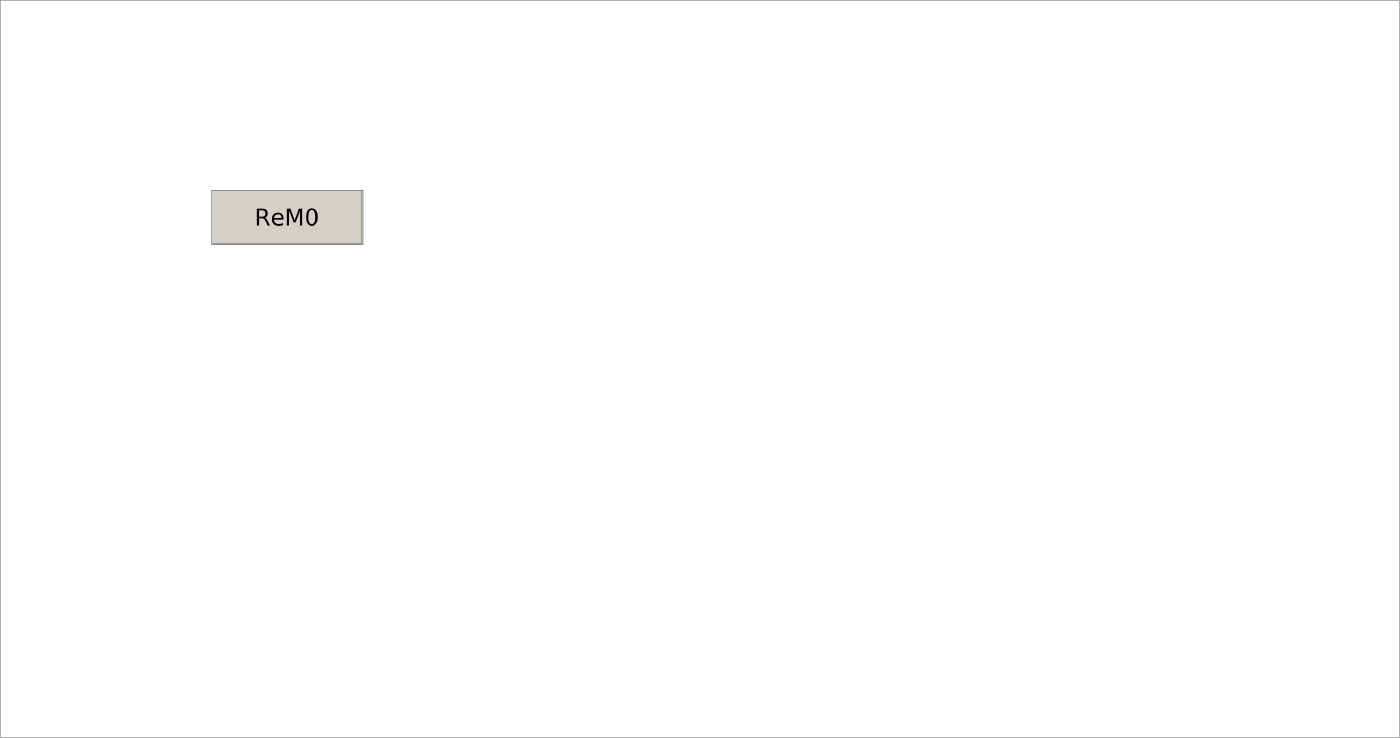
VISUALIZATION visu_Others  // 2048x1080
    Button (309,278 222x80), "ReM0", colour toggle: G_HMI.iReM =0
        p573394764: 16#FF00FF00
        OnMouseDown: execute { G_HMI.iReM  := 0; G_HMI.iMainFrame	:= 0; }
END_VISUALIZATION

(* stored: Version 1.1.0.1, ProductVersion 3.1.4024.12
   Visu visu_Others: Id {5ba4f502-57cb-4741-a8ec-1b5444659dad} *)
